FUNCTION_BLOCK New (* _ *)
  (* Version 2015-09-16 *)
END_FUNCTION_BLOCK
(* other elements stored in the file *)
(* SNS LeftPageBorder=-300.0 RightPageBorder=300.0 *)
